TYPE ST_MachineParameters :
STRUCT
	sSerialNumber			: STRING;
	stAxisM1				: ST_MachineParametersAxis;
	stAxisM2				: ST_MachineParametersAxis;
END_STRUCT
END_TYPE

(* stored: Version 1.1.0.1, ProductVersion 3.1.4024.11
   DUT ST_MachineParameters: Id {c0083ad2-f5f5-462d-a9d5-d9d5037fd6b9} *)
